FUNCTION_BLOCK FB_RANDOM (* Generate a REAL Randomly *)
  (* Standard: 61499-1; Classification: Mathematic; Function: RANDOM; Type: Mathematical function; Description: Copyright (c) 2012 Profactor GmbH This program and the accompanying materials are made available under the terms of the Eclipse Public License 2.0 which is available at https://www.eclipse.org/legal/epl-2.0/ SPDX-License-Identifier: EPL-2.0 *)
  (* Version 1.0, 2012-05-31, Gerhard Ebenhofer, Profactor GmbH *)
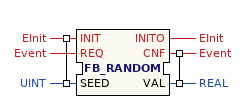
  EVENT_INPUT
    INIT : EInit WITH SEED; (* Initializes the random with the specified seed, if not called the generated values will always be identical *)
    REQ; (* Calculates a new random number between 0 and 1 *)
  END_EVENT
  EVENT_OUTPUT
    INITO : EInit;
    CNF WITH VAL; (* Execution Confirmation *)
  END_EVENT
  VAR_INPUT
    SEED : UINT := 0; (* the seed to initialize the random, a seed of 0 (zero) uses the current systemtime as seed *)
  END_VAR
  VAR_OUTPUT
    VAL : REAL; (* Function output *)
  END_VAR
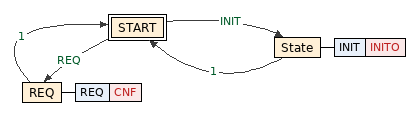
  EC_STATES
    START; (* Initial State *)
    REQ : REQ -> CNF; (* Normal execution *)
    State : INIT -> INITO;
  END_STATES
  EC_TRANSITIONS
    START TO REQ := REQ;
    REQ TO START := 1;
    START TO State := INIT;
    State TO START := 1;
  END_TRANSITIONS
  ALGORITHM INIT IN AnyText: (* ALG *)
// WARNING - Don't forget to add #include <time.h>

if (SEED() == 0) {
  srand( (unsigned int) time(NULL) );
} else {
  srand( SEED() );
}
  END_ALGORITHM
  ALGORITHM REQ IN AnyText: (* Normally executed algorithm *)
VAL() = (TForteFloat) ((rand() % 32767) / 100000.0); // RAND_MAX is a constant defined in <cstdlib>. Its default value may vary between implementations but it is granted to be at least 32767.
  END_ALGORITHM
END_FUNCTION_BLOCK
